(* IEC 61131-3 sources: CodesysTest/export/UN00 - Sharp Bagger/EM02 - Discharge/CM00 - Retracting Load Plate/FB_SimBasicLoadPlate.pou/ReadyToLoad.prop, 1 file *)

(* ---- Get.pm.st ---- *)
(*#-#-#-#-#-#-#-#-#-#---Declaration---#-#-#-#-#-#-#-#-#-#-#-#-#*)

VAR
END_VAR
(*#-#-#-#-#-#-#-#-#-#---Implementation---#-#-#-#-#-#-#-#-#-#-#-#-#*)

ReadyToLoad := beginDischarge.Q;
